// TwinCAT 3 PLC project Examples
// ProgramVersion: 3.1.4023.0
// libraries:
//   tc-tools, * (hganchev)
//   Tc2_MC2, * (Beckhoff Automation GmbH)
//   Tc2_Standard, * (Beckhoff Automation GmbH)
//   Tc2_System, * (Beckhoff Automation GmbH)
//   Tc3_Module, * (Beckhoff Automation GmbH)
// project tree:
//   / PlcTask.TcTTO
//   POUs/Examples/ExportREALData/ ExportRealDataToFile.TcPOU
//   POUs/ MAIN.TcPOU

CONFIGURATION Examples
    RESOURCE PLC ON TwinCAT3
        TASK PlcTask(INTERVAL := T#10ms, PRIORITY := 20);
        PROGRAM MAIN WITH PlcTask : MAIN;
    END_RESOURCE
END_CONFIGURATION

// ---- POUs/MAIN.TcPOU
PROGRAM MAIN
VAR
	axisRef				: AXIS_REF;
	fbAxisControl		: MC_AxisControl;
END_VAR

fbAxisControl(axisRef:= axisRef);

END_PROGRAM

// ---- POUs/Examples/ExportREALData/ExportRealDataToFile.TcPOU
FUNCTION_BLOCK ExportRealDataToFile
VAR_INPUT
	arrREALData				: ARRAY[0..Parameters.iArrayREALSize] OF REAL;
	sFilePath				: STRING(255); // File Path
	bUseTimeStamp 			: BOOL;
	bRoundREALDataValues	: BOOL;
	iRoundingDecIndex		: INT := 2; 
	
	bExport					: BOOL;
END_VAR
VAR_OUTPUT
	bExportDone					: BOOL; // Trigger signal for ExportDone
END_VAR
VAR	
	sInputFilePath			: STRING(255);
	// TimeStamp
	timeStamp				: STRING(255);
	sFilePathPlusTimestamp	: STRING(255);
	fbSysTime   			: FB_LocalSystemTime := ( bEnable := TRUE, dwCycle := 1 );
	
	// Export Data
	fbExport 				: ExportArrayREALDataToTextFile;
	
	i						: INT;
END_VAR

// get system time
fbSysTime();

// use time stamp to file name
IF bUseTimeStamp THEN
	// get time stamp
	timeStamp := F_GET_TIME_STAMP(fbSysTime.systemTime, '_', '_');
	sFilePathPlusTimestamp := INSERT(sFilePath,CONCAT('_',timeStamp),FIND(sFilePath, '.txt') - 1);
	sInputFilePath := sFilePathPlusTimestamp;
ELSE
	sInputFilePath := sFilePath;
END_IF

// round array data values
IF bRoundREALDataValues THEN
	FOR i := 0 TO Parameters.iArrayREALSize DO
		arrREALData[i] := F_ROUND_REAL(arrREALData[i], iRoundingDecIndex);
	END_FOR
END_IF


fbExport(
	arrData:= arrREALData, 
	bExecute:= bExport, 
	bUseTimeStamp:= bUseTimeStamp, 
	sFilePath:= sInputFilePath, 
	bDone=> bExportDone);

END_FUNCTION_BLOCK
